(* IEC 61131-3 sources: Industry-PLC-LLM/data/PLCBEAD_repo/PLCBEAD_PLCEmbed-main/PLC-BEAD/Source/GEB/MS_TO_BFT, 1 file *)

(* ---- MS_TO_BFT.ST ---- *)
FUNCTION MS_TO_BFT:INT

	VAR_INPUT
		MS :	REAL;
	END_VAR

	MS_TO_BFT := REAL_TO_INT(EXPT(MS * 1.196172, 0.666667));

END_FUNCTION

PROGRAM program0
	VAR
		MS :	REAL;

		OUT : INT;
	END_VAR

	OUT := MS_TO_BFT(MS);

END_PROGRAM
